(* PLC project Tc2_Utilities.FB_MemBufferSplit Demo, tc3-libraries-kb TwinCAT 3.1 *)
(* stored: creationDateTime 2026-05-11T00:00:00, modificationDateTime 2026-05-11T00:00:00 *)

PROGRAM P_Demo_FB_MemBufferSplit
  VAR
    fbFB_MemBufferSplit : FB_MemBufferSplit;  (* FB_MemBufferSplit 实例 *)
    eCmd : E_EnumCmdType := eEnumCmd_First;
    pBuffer : POINTER TO BYTE;
    cbBuffer : UDINT;
    cbSize : UDINT;
    bOk : BOOL;
    pSegment : POINTER TO BYTE;
    cbSegment : UDINT;
    bEOS : BOOL;
  END_VAR

// =============================================================================
// 场景：拆通讯协议包。
// 价值：意图清晰。
// 验证：给一段缓冲 + 拆分位置 N，触发后前 N 字节进段 1，剩余进段 2。
// 验证步骤：
//   1. 右键 PLC 项目 → Import PLCopenXML → 选本文件
//   2. 引用 Tc2_Utilities（References → Add library）
//   3. 编译 → 登录 → 运行；按上方『验证』行的指示在线写值观察
// =============================================================================

// 单次完整调用形式（所有 VAR_INPUT 显式赋值）
fbFB_MemBufferSplit(
    eCmd := eCmd,
    pBuffer := pBuffer,
    cbBuffer := cbBuffer,
    cbSize := cbSize,
    bOk => bOk,
    pSegment => pSegment,
    cbSegment => cbSegment,
    bEOS => bEOS
);
END_PROGRAM
